FUNCTION_BLOCK Starting_State_Sample  IMPLEMENTS ITF_State
VAR_INPUT
END_VAR
VAR_OUTPUT
END_VAR
VAR
	pPML_Base : POINTER TO PML_Base;
	_stateMachine : IPmlStateMachine;
	bRun: BOOL;
END_VAR

METHOD Cycle : BOOL
VAR_INPUT
END_VAR
IF bRun THEN
	_stateMachine.SetStateComplete();
	pPML_Base^.SetState(pPML_Base^.execute);
END_IF
END_METHOD

METHOD FB_init : BOOL
VAR_INPUT
	bInitRetains : BOOL; // if TRUE, the retain variables are initialized (warm start / cold start)
	bInCopyCode : BOOL;  // if TRUE, the instance afterwards gets moved into the copy code (online change)
	pPML_Base : POINTER TO PML_Base;
	statemachine : IPmlStateMachine;
END_VAR
_stateMachine := statemachine;
THIS^.pPML_Base := pPML_Base;
END_METHOD

END_FUNCTION_BLOCK

(* stored: Version 1.1.0.1, ProductVersion 3.1.4024.11
   POU Starting_State_Sample: Id {899a86a6-3bd5-45c4-b16c-5661c37404d1}, SpecialFunc None
   Method Cycle: Id {7c853f0a-b4f2-4b83-9f12-9b89748beece}
   Method FB_init: Id {d2223c37-5e4d-4ac6-9d32-ddda32e74881} *)
